// TIA Portal V18 export
TYPE "Processing_ShW"
// stored: IsFailsafeCompliant false
   STRUCT
      Trigger : Bool;
   END_STRUCT;
END_TYPE
